FUNCTION_BLOCK ObserveStack EXTENDS HardwareObservationBase
VAR_INPUT
END_VAR
VAR_OUTPUT
END_VAR
VAR
	m_ptrStack: POINTER TO Stack;
	m_ptrStackWP: POINTER TO xPPUProduct;
END_VAR

METHOD FB_init : BOOL
VAR_INPUT
	bInitRetains : BOOL; // if TRUE, the retain variables are initialized (warm start / cold start)
	bInCopyCode : BOOL;  // if TRUE, the instance afterwards gets moved into the copy code (online change)

	i_ptrStack: POINTER TO Stack;
	i_ptrWP: POINTER TO xPPUProduct;
END_VAR
m_ptrStack := i_ptrStack;
m_ptrStackWP := i_ptrWP;
END_METHOD

METHOD  ResetDefinition : BOOL
VAR_INPUT
END_VAR
;
END_METHOD

(* Update an instance of ProcessState with the part of the process that can be observed by this Hardware Interface. *)
METHOD UpdateProcessObservation : BOOL
VAR_IN_OUT
	io_processState: ProcessState;
END_VAR
io_processState.UpdateState_Binary(EProcessVariables.Stack_WorkpieceAvailable, m_ptrStack^.WPOnTray, i_force := TRUE);
io_processState.UpdateState_Binary(EProcessVariables.Stack_CylinderExtended, m_ptrStack^.o_slidingCylinder.Extended, i_force := TRUE);
io_processState.UpdateState_Binary(EProcessVariables.Stack_CylinderRetracted, m_ptrStack^.o_slidingCylinder.Retracted, i_force := TRUE);

io_processState.UpdateState_Defined(EProcessVariables.Stack_WorkpieceAvailable, TRUE);
io_processState.UpdateState_Defined(EProcessVariables.Stack_CylinderExtended, TRUE);
io_processState.UpdateState_Defined(EProcessVariables.Stack_CylinderRetracted, TRUE);

// update WP info (if there are sensors available), then update the process variables list
m_ptrStackWP^.IsPresent := m_ptrStack^.WPOnTray;
m_ptrStackWP^.IsLight := m_ptrStack^.LightWPOnTray;
m_ptrStackWP^.IsMetal := m_ptrStack^.MetalWPOnTray;
END_METHOD

END_FUNCTION_BLOCK

(* stored: Version 1.1.0.1
   POU ObserveStack: Id {699d7880-46fc-45fa-945d-1111af0fe09e}, SpecialFunc None
   Method FB_init: Id {28d42989-0478-47fa-a8e0-10e62d7763aa}
   Method ResetDefinition: Id {23057aa0-ce57-41cb-bff6-13a68f96659f}
   Method UpdateProcessObservation: Id {63c22b01-f7f9-454f-8201-2ad3fb9c21f9} *)
